// Return TRUE for nIn = Err.End.
// Optionally carries the value over to nOut for further processing.
FUNCTION IsEnd : BOOL
VAR_INPUT
    nIn : Result; // Result variable to check for any non-None value
END_VAR
VAR_OUTPUT
    nOut : Result; // Carries the input value for further use
END_VAR

IsEnd := nIn = Err.End;
nOut := nIn;

END_FUNCTION

(* stored: Version 1.1.0.1
   POU IsEnd: Id {64e2b328-2c41-4ea4-acc1-b6d7b61cfb9d}, SpecialFunc None *)
